(* Logix 5000 project; controller Drives_Line1 1756-L72 rev 20.13; software revision 20.04; part 21 of 21 *)
(* tags used below, declared in another part *)
   Bridle_01 : UDT_Bridle_3M;
   Bridle_02 : UDT_Bridle_2M;
   Bridle_03 : UDT_Bridle_2M;
   Bridle_04 : UDT_Bridle_3M;
   Entry_Accu : UDT_Entry_Accu;
   EntryCtrl : UDT_Control_Zone;
   Exit_Accu : UDT_Exit_Accu;
   ExitCtrl : UDT_Control_Zone;
   ForSimulation : REAL[100];
   MainFltHndler : DINT[11];
   Out_Feedbacks : UDT_Fdbks;
   Out_Status : UDT_Status;
   Pinchroll_1 : UDT_Pinchroll;
   Pinchroll_2 : UDT_Pinchroll;
   Pinchroll_3 : UDT_Pinchroll;
   TM1 : UDT_TM;
   TM2 : UDT_TM;
   TM3 : UDT_TM;
   Unwinder_1 : UDT_Unwinder;
   Unwinder_2 : UDT_Unwinder;
   Winder : UDT_Winder;
   zBridle_01a_EncRes : DINT;
   zBridle_02a_EncRes : DINT;
   zBridle_04a_EncRes : DINT;
   zPinchroll_2_EncRes : DINT;
   zPinchroll_3_EncRes : DINT;
   zSimulation : BOOL;
(* P21_Pinchroll_3, continued *)

ROUTINE R99_To_Master   (* ladder *)
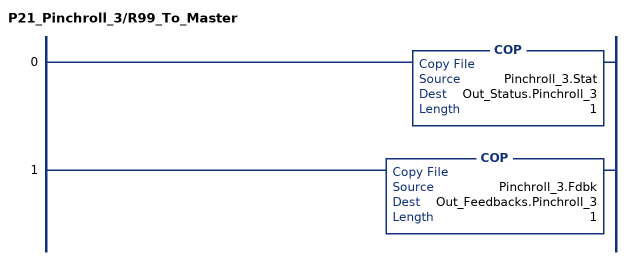
   0: COP(Pinchroll_3.Stat,Out_Status.Pinchroll_3,1);
   1: COP(Pinchroll_3.Fdbk,Out_Feedbacks.Pinchroll_3,1);
END_ROUTINE
END_PROGRAM

PROGRAM P99_FaultHandler   (* main routine R00_Main *)

ROUTINE R00_Main   (* ladder *)
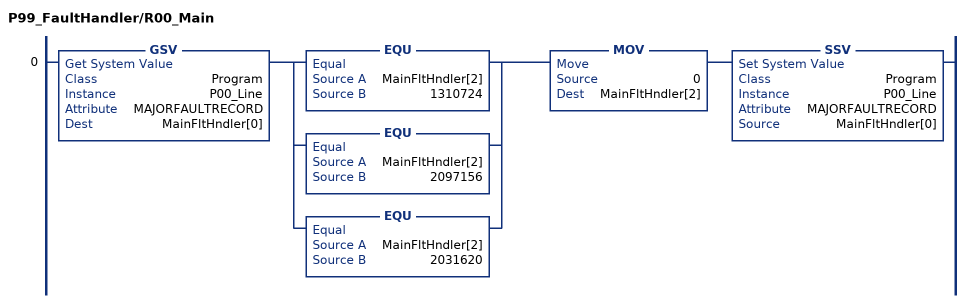
   0: GSV(Program,P00_Line,MAJORFAULTRECORD,MainFltHndler[0])[EQU(MainFltHndler[2],1310724) ,EQU(MainFltHndler[2],2097156) ,EQU(MainFltHndler[2],2031620) ]MOV(0,MainFltHndler[2])SSV(Program,P00_Line,MAJORFAULTRECORD,MainFltHndler[0]);
END_ROUTINE
END_PROGRAM

PROGRAM P99_Simulation   (* main routine R00_Main *)
VAR
   DEDT_01 : DEADTIME := (In := 249.94383, Deadtime := 2.0, Gain := 1.0, RTSTime := 1, Out := 249.93764, DeltaT := 0.05);
   DEDT_TM : REAL[50] := ([0] := 249.94002, [1] := 249.94017, [2] := 249.94032, [3] := 249.94048, [4] := 249.94063, [5] := 249.94078, [6] := 249.94093, [7] := 249.94109, [8] := 249.94124, [9] := 249.94139, [10] := 249.94154, [11] := 249.9417, [12] := 249.94185, [13] := 249.942, [14] := 249.94215, [15] := 249.9423, [16] := 249.94246, [17] := 249.94261, [18] := 249.94276, [19] := 249.94292, [20] := 249.94307, [21] := 249.94322, [22] := 249.94337, [23] := 249.94353, [24] := 249.94368, [25] := 249.93596, [26] := 249.93613, [27] := 249.9363, [28] := 249.93646, [29] := 249.93663, [30] := 249.9368, [31] := 249.93697, [32] := 249.93713, [33] := 249.9373, [34] := 249.93747, [35] := 249.93764, [36] := 249.9378, [37] := 249.93797, [38] := 249.93814, [39] := 249.93831, [40] := 249.93848, [41] := 249.93864, [42] := 249.9388, [43] := 249.93895, [44] := 249.9391, [45] := 249.93925, [46] := 249.9394, [47] := 249.93956, [48] := 249.93971, [49] := 249.93987);
   DIV_02 : FBD_MATH := (SourceA := 38014.367, SourceB := 60.0, Dest := 633.5728);
   DIV_04 : FBD_MATH := (SourceB := 60.0);
   DIV_06 : FBD_MATH := (SourceB := 60.0);
   DIV_07 : FBD_MATH := (SourceA := 43564.844, SourceB := 60.0, Dest := 726.08075);
   DIV_08 : FBD_MATH := (SourceB := 60.0);
   INTG_01 : INTEGRATOR := (In := 3123.2083, IGain := 1.0, RTSTime := 1, Out := 2839203.8, DeltaT := 0.05);
   INTG_02 : INTEGRATOR := (In := 633.5728, IGain := 1.0, RTSTime := 1, Out := 640965.94, DeltaT := 0.05);
   INTG_03 : INTEGRATOR := (In := 726.08075, IGain := 1.0, RTSTime := 1, Out := 728308.06, DeltaT := 0.05);
   INTG_04 : INTEGRATOR := (IGain := 1.0, RTSTime := 1, Out := 233232.61, DeltaT := 0.05);
   INTG_05 : INTEGRATOR := (IGain := 1.0, RTSTime := 1, Out := 112610.086, DeltaT := 0.05);
   INTG_06 : INTEGRATOR := (IGain := 1.0, RTSTime := 1, DeltaT := 0.05);
   INTG_08 : INTEGRATOR := (IGain := 1.0, RTSTime := 1, Out := 252807.27, DeltaT := 0.05);
   LDLG_01 : LEAD_LAG := (In := 249.9518, Lag := 2.5, Gain := 1.0, RTSTime := 1, Out := 249.94383, DeltaT := 0.05);
   LDLG_03 : LEAD_LAG := (Lag := 2.0, Gain := 1.0, RTSTime := 1, Out := 1.0120747, DeltaT := 0.05);
   LDLG_04 : LEAD_LAG := (In := -1.9250553, Lag := 2.0, Gain := 1.0, RTSTime := 1, Out := -1.8826115, DeltaT := 0.05);
   LDLG_05 : LEAD_LAG := (Lag := 2.0, Gain := 1.0, RTSTime := 1, DeltaT := 0.05);
   LDLG_06 : LEAD_LAG := (In := 250.00163, Lag := 2.0, Gain := 1.0, RTSTime := 1, Out := 250.00146, DeltaT := 0.05);
   LDLG_07 : LEAD_LAG := (In := 88.36004, Lag := 2.0, Gain := 1.0, RTSTime := 1, Out := 88.36002, DeltaT := 0.05);
   MUL_01 : FBD_MATH := (SourceA := 37.280552, SourceB := 1024.0, Dest := 38175.285);
   MUL_03 : FBD_MATH := (SourceB := 1024.0);
   MUL_05 : FBD_MATH := (SourceB := 1024.0);
   MUL_06 : FBD_MATH := (SourceA := 42.543793, SourceB := 1024.0, Dest := 43564.844);
   MUL_07 : FBD_MATH := (SourceB := 1024.0);
   SCL_01 : SCALE := (InRawMax := 0.083, InEUMax := 1000.0, Limiting := 1);
   SCL_02 : SCALE := (In := 0.008250054, InRawMax := 0.033, InEUMax := 1000.0, Limiting := 1, Out := 250.00163);
   SCL_03 : SCALE := (InRawMax := 1.0, InRawMin := -1.0, InEUMax := 512000.0, InEUMin := -512000.0, Limiting := 1);
   SCL_06 : SCALE := (In := 0.008248409, InRawMax := 0.033, InEUMax := 1000.0, Out := 249.9518);
   SCL_07 : SCALE := (In := 0.006100016, InRawMax := 1.0, InRawMin := -1.0, InEUMax := 512000.0, InEUMin := -512000.0, Limiting := 1, Out := 3123.2083);
END_VAR

ROUTINE R00_Main   (* ladder *)
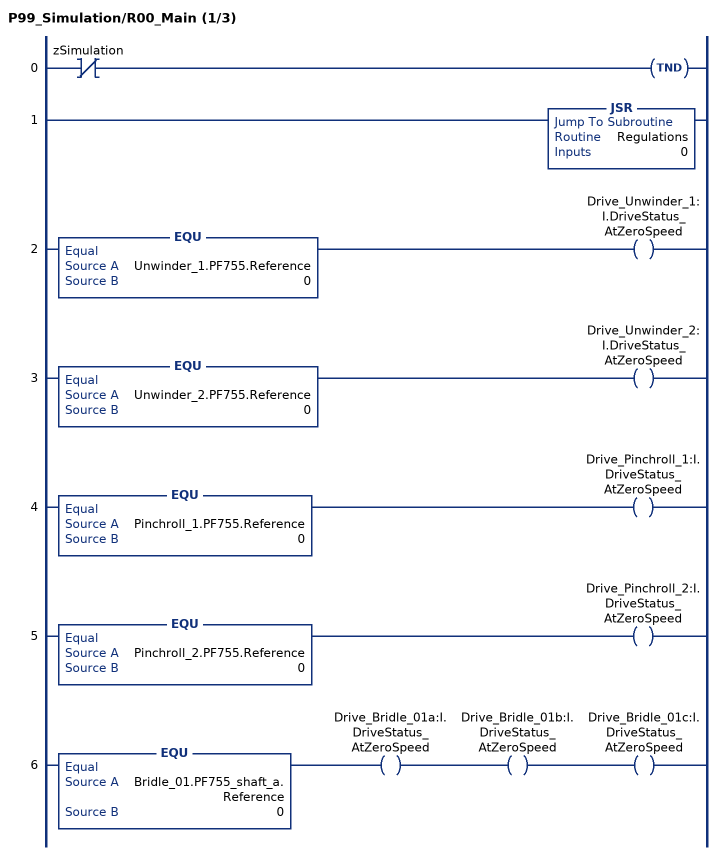
   0: XIO(zSimulation)TND();
   1: JSR(Regulations,0);
   2: EQU(Unwinder_1.PF755.Reference,0)OTE(Drive_Unwinder_1:I.DriveStatus_AtZeroSpeed);
   3: EQU(Unwinder_2.PF755.Reference,0)OTE(Drive_Unwinder_2:I.DriveStatus_AtZeroSpeed);
   4: EQU(Pinchroll_1.PF755.Reference,0)OTE(Drive_Pinchroll_1:I.DriveStatus_AtZeroSpeed);
   5: EQU(Pinchroll_2.PF755.Reference,0)OTE(Drive_Pinchroll_2:I.DriveStatus_AtZeroSpeed);
   6: EQU(Bridle_01.PF755_shaft_a.Reference,0)OTE(Drive_Bridle_01a:I.DriveStatus_AtZeroSpeed)OTE(Drive_Bridle_01b:I.DriveStatus_AtZeroSpeed)OTE(Drive_Bridle_01c:I.DriveStatus_AtZeroSpeed);
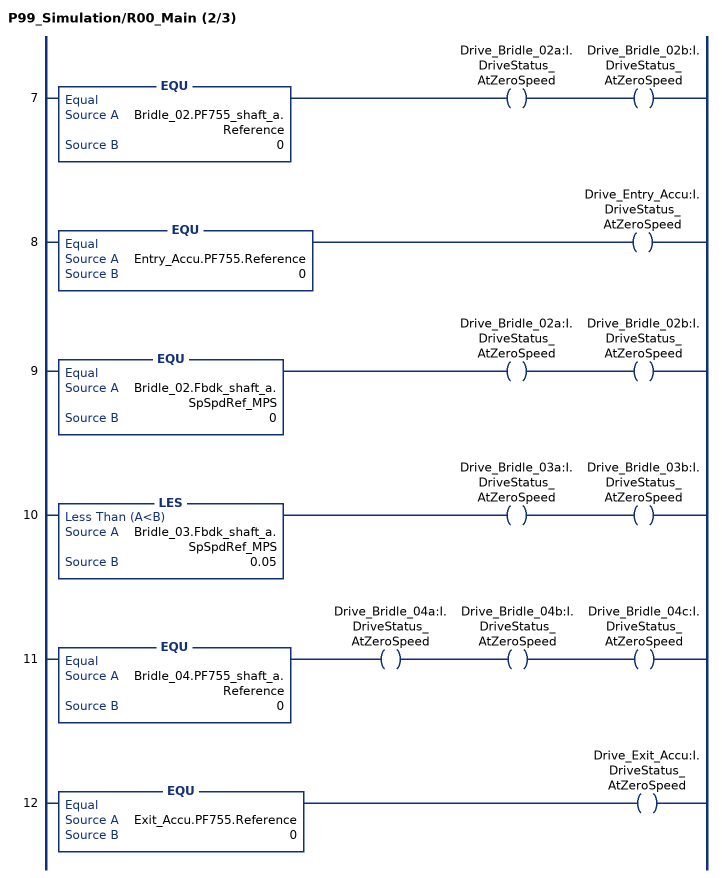
   7: EQU(Bridle_02.PF755_shaft_a.Reference,0)OTE(Drive_Bridle_02a:I.DriveStatus_AtZeroSpeed)OTE(Drive_Bridle_02b:I.DriveStatus_AtZeroSpeed);
   8: EQU(Entry_Accu.PF755.Reference,0)OTE(Drive_Entry_Accu:I.DriveStatus_AtZeroSpeed);
   9: EQU(Bridle_02.Fbdk_shaft_a.SpSpdRef_MPS,0)OTE(Drive_Bridle_02a:I.DriveStatus_AtZeroSpeed)OTE(Drive_Bridle_02b:I.DriveStatus_AtZeroSpeed);
   10: LES(Bridle_03.Fbdk_shaft_a.SpSpdRef_MPS,0.05)OTE(Drive_Bridle_03a:I.DriveStatus_AtZeroSpeed)OTE(Drive_Bridle_03b:I.DriveStatus_AtZeroSpeed);
   11: EQU(Bridle_04.PF755_shaft_a.Reference,0)OTE(Drive_Bridle_04a:I.DriveStatus_AtZeroSpeed)OTE(Drive_Bridle_04b:I.DriveStatus_AtZeroSpeed)OTE(Drive_Bridle_04c:I.DriveStatus_AtZeroSpeed);
   12: EQU(Exit_Accu.PF755.Reference,0)OTE(Drive_Exit_Accu:I.DriveStatus_AtZeroSpeed);
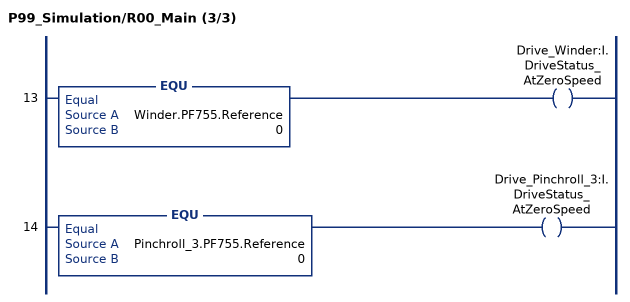
   13: EQU(Winder.PF755.Reference,0)OTE(Drive_Winder:I.DriveStatus_AtZeroSpeed);
   14: EQU(Pinchroll_3.PF755.Reference,0)OTE(Drive_Pinchroll_3:I.DriveStatus_AtZeroSpeed);
END_ROUTINE

ROUTINE Regulations   (* function block diagram *)
   SHEET 1   // Position feedback entry accu
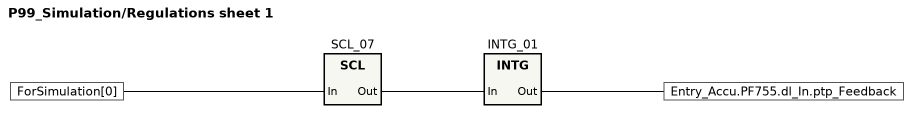
   SCL_07 : SCL(In := ForSimulation[0]);
   INTG_01 : INTG(In := SCL_07.Out);
   Entry_Accu.PF755.dl_In.ptp_Feedback := INTG_01.Out;
   SHEET 2   // Tension feedback entry accu
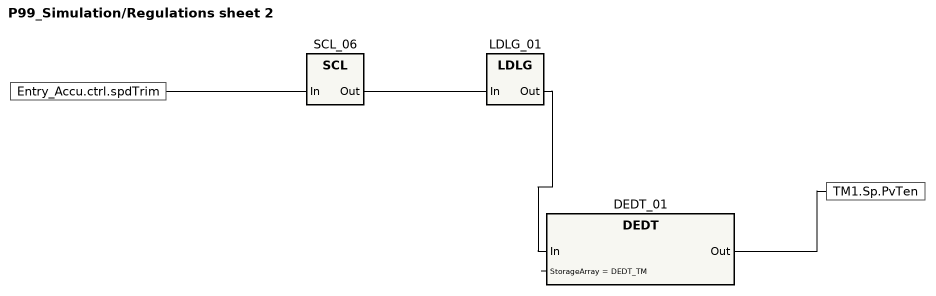
   SCL_06 : SCL(In := Entry_Accu.ctrl.spdTrim);
   LDLG_01 : LDLG(In := SCL_06.Out);
   DEDT_01 : DEDT(In := LDLG_01.Out, StorageArray := DEDT_TM);
   TM1.Sp.PvTen := DEDT_01.Out;
   SHEET 3   // Tension feedback TM2
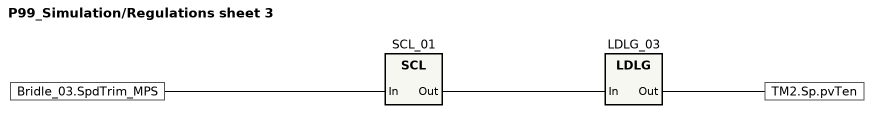
   SCL_01 : SCL(In := Bridle_03.SpdTrim_MPS);
   LDLG_03 : LDLG(In := SCL_01.Out);
   TM2.Sp.pvTen := LDLG_03.Out;
   SHEET 4   // Unwinder 1 & 2 & Winder tension feedback
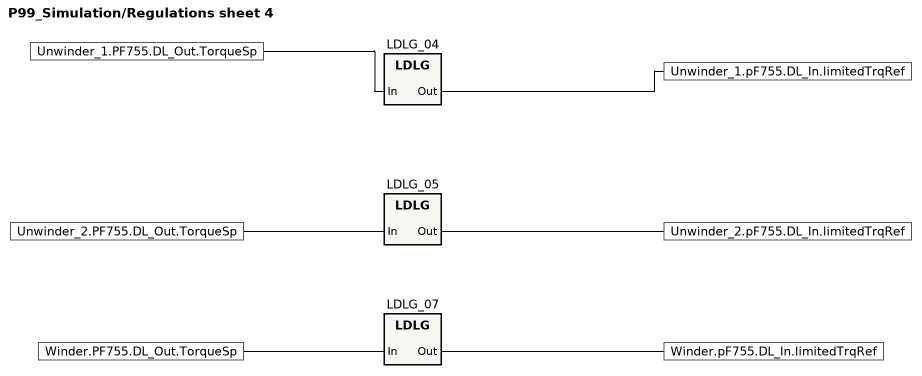
   LDLG_04 : LDLG(In := Unwinder_1.PF755.DL_Out.TorqueSp);
   LDLG_05 : LDLG(In := Unwinder_2.PF755.DL_Out.TorqueSp);
   LDLG_07 : LDLG(In := Winder.PF755.DL_Out.TorqueSp);
   Unwinder_1.pF755.DL_In.limitedTrqRef := LDLG_04.Out;
   Unwinder_2.pF755.DL_In.limitedTrqRef := LDLG_05.Out;
   Winder.pF755.DL_In.limitedTrqRef := LDLG_07.Out;
   SHEET 5   // Bridle 01 PTP feedback
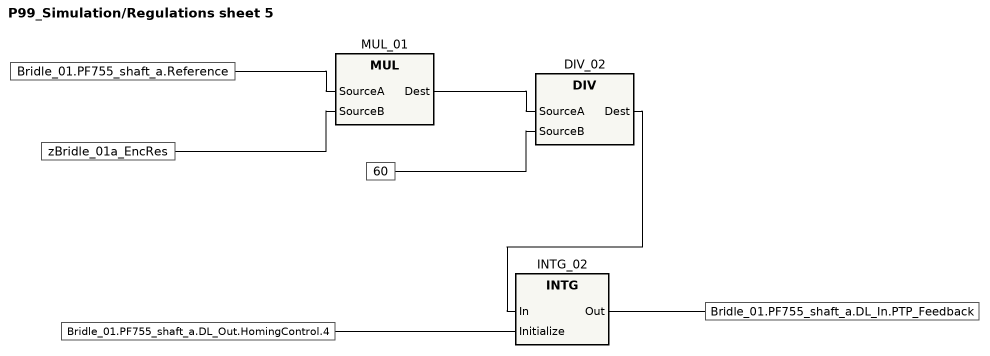
   MUL_01 : MUL(SourceA := Bridle_01.PF755_shaft_a.Reference, SourceB := zBridle_01a_EncRes);
   DIV_02 : DIV(SourceA := MUL_01.Dest, SourceB := 60);
   INTG_02 : INTG(In := DIV_02.Dest, Initialize := Bridle_01.PF755_shaft_a.DL_Out.HomingControl.4);
   Bridle_01.PF755_shaft_a.DL_In.PTP_Feedback := INTG_02.Out;
   SHEET 6   // Pinchroll 2 & 3 feedback
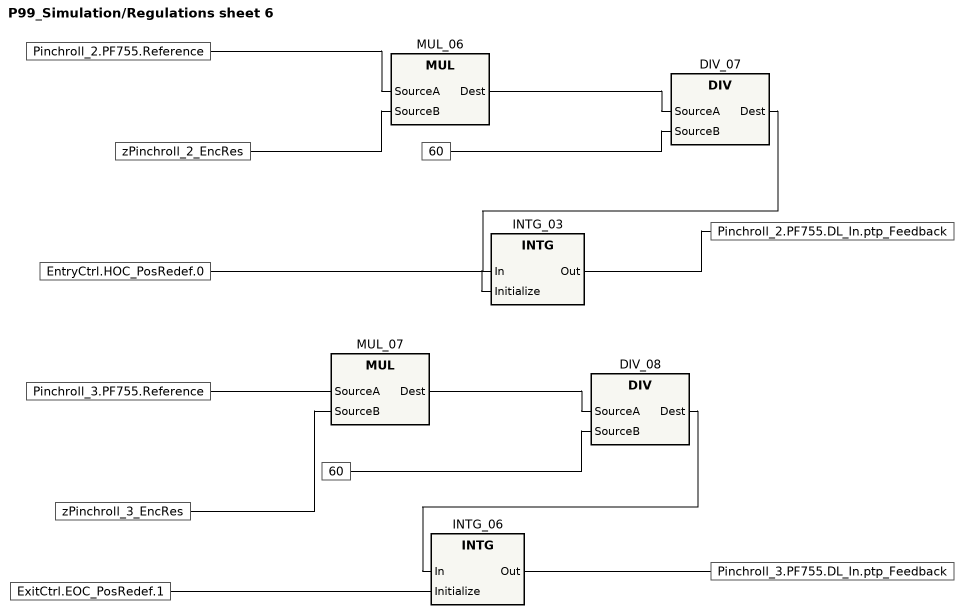
   MUL_07 : MUL(SourceA := Pinchroll_3.PF755.Reference, SourceB := zPinchroll_3_EncRes);
   MUL_06 : MUL(SourceA := Pinchroll_2.PF755.Reference, SourceB := zPinchroll_2_EncRes);
   DIV_08 : DIV(SourceA := MUL_07.Dest, SourceB := 60);
   INTG_06 : INTG(In := DIV_08.Dest, Initialize := ExitCtrl.EOC_PosRedef.1);
   DIV_07 : DIV(SourceA := MUL_06.Dest, SourceB := 60);
   INTG_03 : INTG(In := DIV_07.Dest, Initialize := EntryCtrl.HOC_PosRedef.0);
   Pinchroll_2.PF755.DL_In.ptp_Feedback := INTG_03.Out;
   Pinchroll_3.PF755.DL_In.ptp_Feedback := INTG_06.Out;
   SHEET 7   // Tension feedback TM3
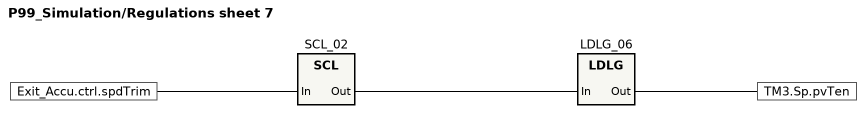
   SCL_02 : SCL(In := Exit_Accu.ctrl.spdTrim);
   LDLG_06 : LDLG(In := SCL_02.Out);
   TM3.Sp.pvTen := LDLG_06.Out;
   SHEET 8   // Position feedback exit accu
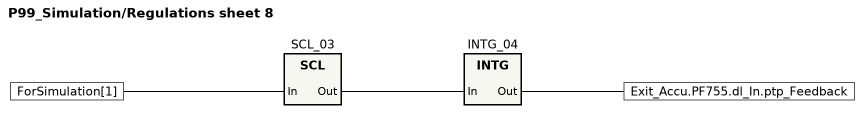
   SCL_03 : SCL(In := ForSimulation[1]);
   INTG_04 : INTG(In := SCL_03.Out);
   Exit_Accu.PF755.dl_In.ptp_Feedback := INTG_04.Out;
   SHEET 9   // Bridle 04 pos feedback
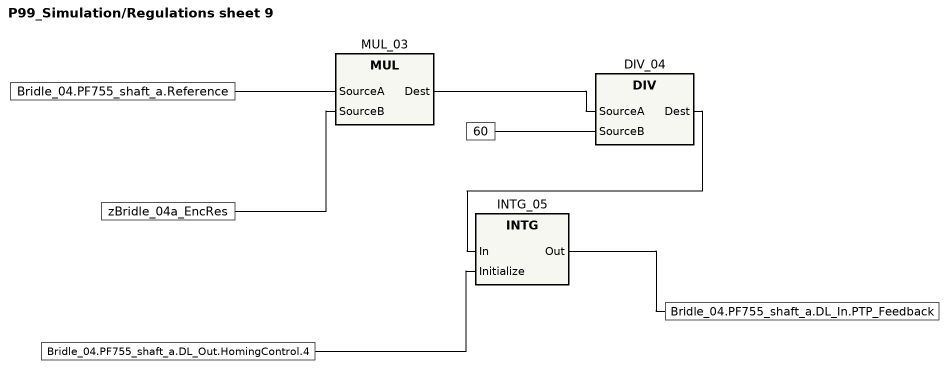
   MUL_03 : MUL(SourceA := Bridle_04.PF755_shaft_a.Reference, SourceB := zBridle_04a_EncRes);
   DIV_04 : DIV(SourceA := MUL_03.Dest, SourceB := 60);
   INTG_05 : INTG(In := DIV_04.Dest, Initialize := Bridle_04.PF755_shaft_a.DL_Out.HomingControl.4);
   Bridle_04.PF755_shaft_a.DL_In.PTP_Feedback := INTG_05.Out;
   SHEET 10   // Bridle 02 pos feedback
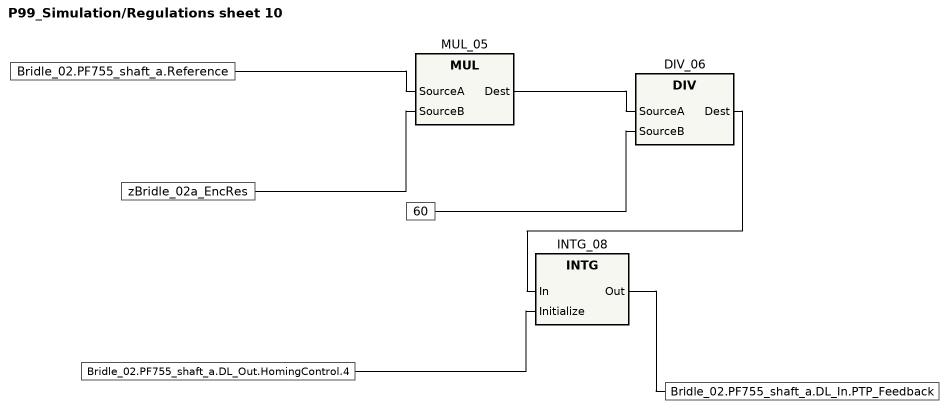
   MUL_05 : MUL(SourceA := Bridle_02.PF755_shaft_a.Reference, SourceB := zBridle_02a_EncRes);
   DIV_06 : DIV(SourceA := MUL_05.Dest, SourceB := 60);
   INTG_08 : INTG(In := DIV_06.Dest, Initialize := Bridle_02.PF755_shaft_a.DL_Out.HomingControl.4);
   Bridle_02.PF755_shaft_a.DL_In.PTP_Feedback := INTG_08.Out;
END_ROUTINE
END_PROGRAM
